# EPICS substitutions: db/Beckhoff_3XXX/ecmcEL3632_s50.substitutions
file "ecmcEcSlave.template"
{
  pattern {}
          {}
}

file "ecmcEL3632-chX.template"
{
  pattern {CH_ID, DTYP,             FTVL,  NELM}
          {1,     asynInt16ArrayIn, SHORT, 50  }
          {2,     asynInt16ArrayIn, SHORT, 50  }
}
